TYPE "TAx_Config"
VERSION : 0.1
// Block: TAx_Config
   STRUCT
      Simulation : Bool;
      PowerOffDelay : Time;
      PowerStartMode : Int;
      PowerStopMode : Int;
   END_STRUCT;

END_TYPE
